// TIA Portal V19 export
TYPE "LEXCHANGETRAY_typeSr1000ProfinetTelegram_completionStatusBits"
// stored: Access Published
   STRUCT
      statusByte : Byte;
      readComplete : Bool;
      presetComplete : Bool;
      registerPresetComplete : Bool;
      tuneComplete : Bool;
      extRequestComplete : Bool;
   END_STRUCT;
END_TYPE
